PROGRAM MAIN_1
VAR
END_VAR

END_PROGRAM

(* stored: Version 1.1.0.1, ProductVersion 3.1.4024.16
   POU MAIN_1: Id {436d51fb-b8cc-43d1-95f5-f2c51dd53cc6}, SpecialFunc None *)
